FUNCTION_BLOCK FB_EventPublisher IMPLEMENTS I_EventPublisher
VAR
	raiseEvent						: BOOL;
	_event							: INT;
	_eventPrev						: INT;
	
	publisher						: FB_Observable;	
END_VAR

IF _eventPrev <> _event 			THEN
	publisher.notify();
	_eventPrev := _event;
END_IF

METHOD attach : BOOL
VAR_INPUT
	observer			: I_Observer;
END_VAR
attach := publisher.attach(observer);
END_METHOD

PROPERTY PUBLIC changeEvent : int
SET
// IMPLEMENTED ONLY FOR TESTING PURPOSES
VAR
END_VAR
_event := changeEvent;
END_SET
END_PROPERTY

METHOD detach : BOOL
VAR_INPUT
	observer	: I_Observer;
END_VAR
detach := publisher.detach(observer);
END_METHOD

// IMPLEMENTED ONLY FOR TESTING PURPOSES
PROPERTY event : int
GET
event := _event;
END_GET
END_PROPERTY

PROPERTY NoOfAttachedObservers : int
GET
NoOfAttachedObservers := publisher.NoOfAttachedObservers;
END_GET
END_PROPERTY

END_FUNCTION_BLOCK

(* stored: Version 1.1.0.1, ProductVersion 3.1.4024.11
   POU FB_EventPublisher: Id {270e0f21-f10c-4d6e-aaab-748f1b75e82c}, SpecialFunc None
   Method attach: Id {ab4ff1ed-f2e9-459d-bd43-c6901c9fa429}
   Property changeEvent: Id {05b37224-02c8-4354-b619-b3cf8f6eb51f}
   Set Set: Id {eda01090-ae55-40a9-bf93-25e50f34c0d7}
   Method detach: Id {0aef42ef-b37c-48ca-9ad5-1143c99045a0}
   Property event: Id {5a53bf6d-f733-4ff7-bc62-c7e9a7ce7ec4}
   Get Get: Id {cdadf8c7-7fab-4fb4-84ee-b1e660efac40}
   Property NoOfAttachedObservers: Id {e1a94e9e-c654-4b44-b5b2-c1d8baedd47d}
   Get Get: Id {f57f8ef9-a1c0-4e55-8245-2af669fb7a07} *)
